// TIA Portal V18 export
// export: Created 2026-03-12T16:04:36.0691038Z, ExportSetting WithDefaults, DisplayName Totally Integrated Automation Portal, DisplayVersion V18 Update 5, DisplayName TIA Portal Openness, DisplayVersion V18 Update 5, DisplayName TIA Portal Version Control Interface, DisplayVersion V18, DisplayName SINAMICS Startdrive Advanced, DisplayVersion V18, DisplayName SINAMICS Startdrive G130, G150, S120, S150, SINAMICS MV, S210, DisplayVersion V18, DisplayName SINAMICS Startdrive G110M, G120, G120C, G120D, G120P, G115D, DisplayVersion V18, DisplayName STEP 7 Professional, DisplayVersion V18 Update 5, DisplayName STEP 7 Safety, DisplayVersion V18, DisplayName WinCC Professional, DisplayVersion V18 Update 5
FUNCTION_BLOCK "FB PROCESSO_ALTERNANCIA_PRINCIPAL_RESERVA"   // FB39, LAD
{ S7_Optimized_Access := 'TRUE' }
VERSION : 0.1
// stored: AutoNumber true, IsIECCheckEnabled false, IsRetainMemResEnabled false, MemoryReserve 100, SetENOAutomatically false, UDAEnableTagReadback false
   VAR_INPUT
      INPUT_HABILITA_PAR : Bool;
      INPUT_REMOTO_AUTO_A : Bool;
      INPUT_REMOTO_AUTO_B : Bool;
      INPUT_COMANDO_ALTERNANCIA_ATIVO : Bool;
      INPUT_FALHA_BOMBA_A : Bool;
      INPUT_FALHA_BOMBA_B : Bool;
      INPUT_CADASTRO_TEMPO_LIGADO_A : Real;
      INPUT_CADASTRO_TEMPO_LIGADO_B : Real;
   END_VAR
   VAR_OUTPUT
      HORA_ALTERNANCIA_A : Real;
      HORA_ALTERNANCIA_B : Real;
      LIGA_ALTERNANCIA_A { ExternalAccessible := 'False'; ExternalVisible := 'False'; ExternalWritable := 'False'} : Bool;
      LIGA_ALTERNANCIA_B { ExternalAccessible := 'False'; ExternalVisible := 'False'; ExternalWritable := 'False'} : Bool;
   END_VAR
   VAR
      "FB CONTADOR_A" { S7_SetPoint := 'True'} : "FB CONTADOR";
      "FB CONTADOR_B" { S7_SetPoint := 'True'} : "FB CONTADOR";
   END_VAR
   VAR_TEMP
      "ALTERNANCIA_ATIVA_A_&_B" : Bool;
   END_VAR
   VAR_TEMP   // added for the SCL form of the ladder/FBD networks
      _w1 : Bool;
   END_VAR
BEGIN

REGION Network 1: Alternância/Rotatividade de bomba Principal
   // Conforme alternância habilitada, a bomba principal e reserva trabalharão intercaladas baseando-se no tempos cadastrados pela operação.
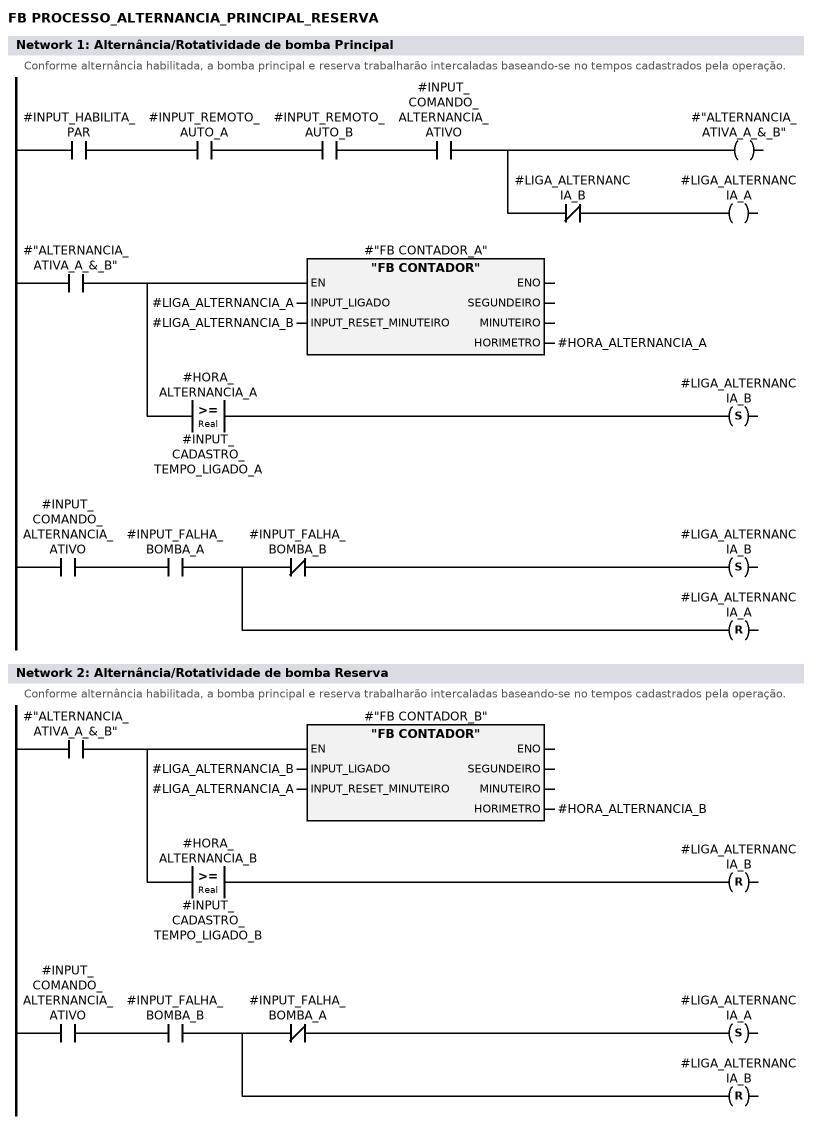
   RUNG wire#powerrail
      Contact( #INPUT_HABILITA_PAR )
      Contact( #INPUT_REMOTO_AUTO_A )
      Contact( #INPUT_REMOTO_AUTO_B )
      Contact( #INPUT_COMANDO_ALTERNANCIA_ATIVO )
      wire#w1
      Coil( #"ALTERNANCIA_ATIVA_A_&_B" )
   END_RUNG
   RUNG wire#w1
      I_Contact( #LIGA_ALTERNANCIA_B )
      Coil( #LIGA_ALTERNANCIA_A )
   END_RUNG
   RUNG wire#powerrail
      Contact( #"ALTERNANCIA_ATIVA_A_&_B" )
      wire#w2
      #"FB CONTADOR_A"(INPUT_LIGADO := #LIGA_ALTERNANCIA_A, INPUT_RESET_MINUTEIRO := #LIGA_ALTERNANCIA_B, SEGUNDEIRO =>, MINUTEIRO =>, HORIMETRO => #HORA_ALTERNANCIA_A)
   END_RUNG
   RUNG wire#w2
      { S7_Templates := "SrcType := Real" } GE_Contact(in1 := #HORA_ALTERNANCIA_A, in2 := #INPUT_CADASTRO_TEMPO_LIGADO_A)
      S_Coil( #LIGA_ALTERNANCIA_B )
   END_RUNG
   RUNG wire#powerrail
      Contact( #INPUT_COMANDO_ALTERNANCIA_ATIVO )
      Contact( #INPUT_FALHA_BOMBA_A )
      wire#w3
      I_Contact( #INPUT_FALHA_BOMBA_B )
      S_Coil( #LIGA_ALTERNANCIA_B )
   END_RUNG
   RUNG wire#w3
      R_Coil( #LIGA_ALTERNANCIA_A )
   END_RUNG
   // the same network as SCL:
   #"ALTERNANCIA_ATIVA_A_&_B" := #INPUT_HABILITA_PAR AND #INPUT_REMOTO_AUTO_A AND #INPUT_REMOTO_AUTO_B AND #INPUT_COMANDO_ALTERNANCIA_ATIVO;
   #LIGA_ALTERNANCIA_A := #"ALTERNANCIA_ATIVA_A_&_B" AND NOT #LIGA_ALTERNANCIA_B;
   IF #"ALTERNANCIA_ATIVA_A_&_B" THEN
       #"FB CONTADOR_A"(INPUT_LIGADO := #LIGA_ALTERNANCIA_A,   // "FB CONTADOR"
                        INPUT_RESET_MINUTEIRO := #LIGA_ALTERNANCIA_B,
                        HORIMETRO => #HORA_ALTERNANCIA_A);
   END_IF;
   IF #"ALTERNANCIA_ATIVA_A_&_B" AND (#HORA_ALTERNANCIA_A >= #INPUT_CADASTRO_TEMPO_LIGADO_A) THEN
       #LIGA_ALTERNANCIA_B := TRUE;
   END_IF;
   #_w1 := #INPUT_COMANDO_ALTERNANCIA_ATIVO AND #INPUT_FALHA_BOMBA_A;
   IF #_w1 AND NOT #INPUT_FALHA_BOMBA_B THEN #LIGA_ALTERNANCIA_B := TRUE; END_IF;
   IF #_w1 THEN #LIGA_ALTERNANCIA_A := FALSE; END_IF;
END_REGION

REGION Network 2: Alternância/Rotatividade de bomba Reserva
   // Conforme alternância habilitada, a bomba principal e reserva trabalharão intercaladas baseando-se no tempos cadastrados pela operação.
   RUNG wire#powerrail
      Contact( #"ALTERNANCIA_ATIVA_A_&_B" )
      wire#w1
      #"FB CONTADOR_B"(INPUT_LIGADO := #LIGA_ALTERNANCIA_B, INPUT_RESET_MINUTEIRO := #LIGA_ALTERNANCIA_A, SEGUNDEIRO =>, MINUTEIRO =>, HORIMETRO => #HORA_ALTERNANCIA_B)
   END_RUNG
   RUNG wire#w1
      { S7_Templates := "SrcType := Real" } GE_Contact(in1 := #HORA_ALTERNANCIA_B, in2 := #INPUT_CADASTRO_TEMPO_LIGADO_B)
      R_Coil( #LIGA_ALTERNANCIA_B )
   END_RUNG
   RUNG wire#powerrail
      Contact( #INPUT_COMANDO_ALTERNANCIA_ATIVO )
      Contact( #INPUT_FALHA_BOMBA_B )
      wire#w2
      I_Contact( #INPUT_FALHA_BOMBA_A )
      S_Coil( #LIGA_ALTERNANCIA_A )
   END_RUNG
   RUNG wire#w2
      R_Coil( #LIGA_ALTERNANCIA_B )
   END_RUNG
   // the same network as SCL:
   IF #"ALTERNANCIA_ATIVA_A_&_B" THEN
       #"FB CONTADOR_B"(INPUT_LIGADO := #LIGA_ALTERNANCIA_B,   // "FB CONTADOR"
                        INPUT_RESET_MINUTEIRO := #LIGA_ALTERNANCIA_A,
                        HORIMETRO => #HORA_ALTERNANCIA_B);
   END_IF;
   IF #"ALTERNANCIA_ATIVA_A_&_B" AND (#HORA_ALTERNANCIA_B >= #INPUT_CADASTRO_TEMPO_LIGADO_B) THEN
       #LIGA_ALTERNANCIA_B := FALSE;
   END_IF;
   #_w1 := #INPUT_COMANDO_ALTERNANCIA_ATIVO AND #INPUT_FALHA_BOMBA_B;
   IF #_w1 AND NOT #INPUT_FALHA_BOMBA_A THEN #LIGA_ALTERNANCIA_A := TRUE; END_IF;
   IF #_w1 THEN #LIGA_ALTERNANCIA_B := FALSE; END_IF;
END_REGION
END_FUNCTION_BLOCK
